{attribute 'pack_mode' := '1'}
TYPE
CT_Shuttle_BR_to_Tc_u :
UNION
    asStruct : ARRAY[1..20] OF CT_Shuttle_BR_to_Tc_t;
    asArray  : ARRAY[0..20 * SIZEOF(CT_Shuttle_BR_to_Tc_t) - 1] OF USINT;
END_UNION
END_TYPE

(* stored: Version 1.1.0.1, ProductVersion 3.1.4024.6
   DUT CT_Shuttle_BR_to_Tc_u: Id {7b704f7b-f9ed-46d6-bd04-74224a79cee2} *)
